FUNCTION_BLOCK Signal_Tests EXTENDS FB_TestSuite
VAR_INPUT
    delta : LREAL := 1E-5;
END_VAR

OnlyMeasurementShouldReturnSameValue();
TakeDerivativeOfMeasurement();
ApplyIirFilterOnSignal();

METHOD ApplyIirFilterOnSignal
VAR_INST
    signal : Signal;
    actual : LREAL;
END_VAR
TEST('ApplyIirFilterOnSignal');

signal.Update(value:=1.4).Iir(decay:=0.5);
AssertEquals_LREAL(Expected:=0.7, Actual:=signal.Out, Delta:=delta, Message:='Output not correct');

actual := signal.Update(value:=8.6).Iir(decay:=0.5).Out;
AssertEquals_LREAL(Expected:=4.65, Actual:=actual, Delta:=delta, Message:='Output not correct');

TcUnit.TEST_FINISHED();
END_METHOD

METHOD OnlyMeasurementShouldReturnSameValue : LREAL
VAR_INST
    signal : Signal;
END_VAR
TEST('OnlyMeasurementShouldReturnSameValue');

signal.Update(value:=1.23);

AssertEquals_LREAL(
    Expected:=1.23,
    Actual:=signal.Out,
    Delta:=delta,
    Message:='Output not correct'
);

TcUnit.TEST_FINISHED();
END_METHOD

METHOD TakeDerivativeOfMeasurement : LREAL
VAR_INST
    signal : Signal;
    actual : LREAL;
END_VAR
TEST('TakeDerivativeOfMeasurement');

actual := signal.Update(value:=1).Differentiate(deltaTime:=1).Out;
AssertEquals_LREAL(
    Expected:=0,
    Actual:=actual,
    Delta:=delta,
    Message:='Derivative after first step not correct'
);

actual := signal.Update(value:=2).Differentiate(deltaTime:=1).Out;
AssertEquals_LREAL(
    Expected:=1,
    Actual:=actual,
    Delta:=delta,
    Message:='Derivative after second step not correct'
);

TcUnit.TEST_FINISHED();
END_METHOD

END_FUNCTION_BLOCK

(* stored: Version 1.1.0.1, ProductVersion 3.1.4024.12
   POU Signal_Tests: Id {7510fb77-c446-4546-9f01-f98754dd3158}, SpecialFunc None
   Method ApplyIirFilterOnSignal: Id {323ff59c-a918-4020-b67e-8db4e2ccd0a4}
   Method OnlyMeasurementShouldReturnSameValue: Id {8a4d1f9e-aae0-4653-b470-003878844f12}
   Method TakeDerivativeOfMeasurement: Id {13d21456-2617-4e90-89f6-0d15220be6a8} *)
